FUNCTION_BLOCK Composite (* Composite Function Block Type *)
  (* Standard: 61499-2 *)
  (* Version 0.2, 2003-12-05, JHC, Rockwell Automation, Renamed from NEWCOMPFB. *)
  (* Version 0.1, 2002-01-08, JHC, Rockwell Automation, Added DLY FB as example. *)
  (* Version 0.0, 2000-05-27, JHC, Rockwell Automation *)
  (* Compiler header: package fb.rt.vhmi;import fb.rt.visual.*; *)
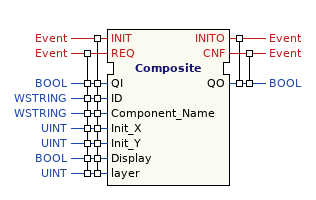
  EVENT_INPUT
    INIT WITH QI, ID, Component_Name, Init_X, Init_Y, Display, layer; (* Initialization Request *)
    REQ WITH QI, ID, Component_Name, Init_X, Init_Y, Display, layer; (* Normal Execution Request *)
  END_EVENT
  EVENT_OUTPUT
    INITO WITH QO; (* Initialization Confirm *)
    CNF WITH QO; (* Execution Confirmation *)
  END_EVENT
  VAR_INPUT
    QI : BOOL; (* Input event qualifier *)
    ID : WSTRING;
    Component_Name : WSTRING;
    Init_X : UINT;
    Init_Y : UINT;
    Display : BOOL;
    layer : UINT;
  END_VAR
  VAR_OUTPUT
    QO : BOOL; (* Output event qualifier *)
  END_VAR
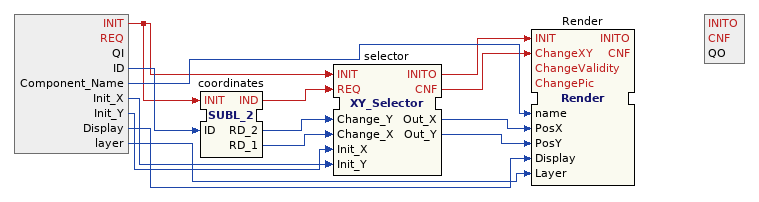
  FBS
    Render : Render;
    coordinates : SUBL_2;
    selector : XY_Selector;
  END_FBS
  EVENT_CONNECTIONS
    INIT TO coordinates.INIT;
    INIT TO selector.INIT;
    selector.INITO TO Render.INIT;
    selector.CNF TO Render.ChangeXY;
    coordinates.IND TO selector.REQ;
  END_CONNECTIONS
  DATA_CONNECTIONS
    coordinates.RD_2 TO selector.Change_Y;
    coordinates.RD_1 TO selector.Change_X;
    selector.Out_X TO Render.PosX;
    selector.Out_Y TO Render.PosY;
    ID TO coordinates.ID;
    Init_X TO selector.Init_X;
    Init_Y TO selector.Init_Y;
    Component_Name TO Render.name;
    layer TO Render.Layer;
    Display TO Render.Display;
  END_CONNECTIONS
END_FUNCTION_BLOCK
